{attribute addProperty BoxType "EL3681-0000-0017"}
{attribute addProperty Id "SAI_InputsAT %I*SAI_Inputs_C1A1928F4860SAI_RangeAT %I*SAI_Range_BF31F39A1620SAI_Range_1AT %Q*SAI_Range_E3AE57CD1620WcStateAT %I*WcState_98A4DF7520.250InfoDataAT %I*InfoData_BC63D37F80100"}
{attribute addProperty CRC "103159124"}
{attribute addProperty SizeInBites "162"}
{attribute addProperty SizeInBytes "20.25"}
TYPE EL3681_0CFA3F61 :
STRUCT
	{attribute addProperty Name "SAI_Inputs"}
	SAI_Inputs : SAI_Inputs_C1A1928F;
	{attribute addProperty Name "SAI_Range"}
	SAI_Range : SAI_Range_BF31F39A;
	{attribute addProperty Name "SAI_Range_1"}
	SAI_Range_1 : SAI_Range_E3AE57CD;
	{attribute addProperty Name "WcState"}
	WcState : WcState_98A4DF75;
	{attribute addProperty Name "InfoData"}
	InfoData : InfoData_BC63D37F;
END_STRUCT
END_TYPE

(* stored: Version 1.2.0.0, ProductVersion 3.1.4024.9
   DUT EL3681_0CFA3F61: Id {1fe40176-a9c1-40d7-ab48-d74be09c9c64} *)
